/// Implicitly generated code : DO NOT EDIT!!!
/// Checks subrange value. If value is outside [lower,upper], it is set to the closer bound and reports the error.
{attribute 'check_range_signed' := ''}
{attribute 'no_check' := ''}
FUNCTION CheckRangeSigned : DINT
VAR_INPUT
	value: DINT;
	lower: DINT;
	upper: DINT;
END_VAR

// align to bounds 
CheckRangeSigned := MIN( upper, MAX( lower, value ));

// if value changed, report error
IF CheckRangeSigned <> value THEN
	GVL_Supervision.aCodeErr[eCodeError_rangeSigned] := TRUE;
END_IF

END_FUNCTION

(* stored: Version 1.1.0.1, ProductVersion 3.1.4022.9
   POU CheckRangeSigned: Id {f1486e31-18e3-4793-9686-f4910b4a9b0b}, SpecialFunc None *)
